Fanuc KAREL source: ko00087.KL

-- PROVISIONAL review KL for V1013-1; original PC SHA256 06d639d692e2a68c36d15cf39e4d2a87f66d9a266537585149bade8206178a84
-- Incomplete behavior may be omitted. Consult companion uncertainty JSON. Do not deploy.
PROGRAM KO00087
%NOLOCKGROUP
BEGIN
  -- UNRESOLVED_PC offsets 5-12; opcodes 9D,23
  -- UNRESOLVED_PC offsets 17-69; opcodes 27,27,49,7E,AD,27,49,7E,AD,22,31,7E,4A
  -- UNRESOLVED_PC offsets 74-78; opcodes 7F
END KO00087
